// TIA Portal V19 export
TYPE "C402_STU_IF_AFS_TYPIC"
   STRUCT
      STU_RES { ExternalAccessible := 'False'; ExternalVisible := 'False'; ExternalWritable := 'False'} : Bool;   // True = reset noodstop kring False = geen sturing
   END_STRUCT;
END_TYPE
